{attribute 'monitoring':='call'}
FUNCTION_BLOCK SlitterMainOperatorPanel

VAR
	
	StartPB		:		NormallyOpenPushButton;
	StopPB		:		NormallyClosePushButton;
	
	StartLight	:		Light;
	StopLight	:		Light;

END_VAR

METHOD PUBLIC StartLightOff : BOOL
VAR_INPUT
END_VAR
StartLight.Off();
END_METHOD

METHOD PUBLIC StartLightOn : BOOL
VAR_INPUT
END_VAR
StartLight.On();
END_METHOD

PROPERTY PUBLIC StartPressed : Bool
GET
StartPressed := StartPB;
END_GET
END_PROPERTY

PROPERTY PUBLIC StartReleased : Bool
GET
StartReleased := NOT StartPressed;
END_GET
END_PROPERTY

METHOD PUBLIC StopLightOff : BOOL
VAR_INPUT
END_VAR
StopLight.Off();
END_METHOD

METHOD PUBLIC StopLightOn : BOOL
VAR_INPUT
END_VAR
StopLight.On();
END_METHOD

PROPERTY PUBLIC StopPressed : Bool
GET
StopPressed := Not StopPB;
END_GET
END_PROPERTY

PROPERTY PUBLIC StopReleased : Bool
GET
StopPressed := Not StopPressed;
END_GET
END_PROPERTY

END_FUNCTION_BLOCK

(* stored: Version 1.1.0.1, ProductVersion 3.1.4024.12
   POU SlitterMainOperatorPanel: Id {8c1fe4af-6777-479f-a0c2-4bd793a745fe}, SpecialFunc None
   Method StartLightOff: Id {2708ce47-e44d-4f2c-9c52-ae80bc07d877}
   Method StartLightOn: Id {1c63e6e5-e132-4e8c-9ee2-073f7e543e44}
   Property StartPressed: Id {4c484f6d-1915-48ba-a5b1-40543bd04621}
   Get Get: Id {02f7aa8f-dfcd-45c6-92fa-1b4bf9beedc3}
   Property StartReleased: Id {31f7ee6c-7352-4a7f-abb6-8d0f67a4f4e5}
   Get Get: Id {2e5a12d9-9db5-460a-83cf-8bd88952a8db}
   Method StopLightOff: Id {f1ea3524-7341-4c87-8ac1-279119b14dbc}
   Method StopLightOn: Id {357b58b4-6586-4552-9c1a-d33de473ab64}
   Property StopPressed: Id {86cd4ebf-9654-4a7a-a02f-d263ec6e9149}
   Get Get: Id {39f5b4ba-a192-4107-8a03-9ad5aba3a4f3}
   Property StopReleased: Id {a959fde0-2f50-4bdf-b9f8-d993972731d7}
   Get Get: Id {52a16103-10c4-4b8f-a8d1-9a40bdc5eb4b} *)
